FUNCTION RFID_Get_String : Buffer_Error
VAR_INPUT
	Data : REFERENCE TO RFID_Tag_Data;
	Num : USINT; 
END_VAR
VAR_IN_OUT
	Out : STRING[8];
END_VAR

RFID_Get_String := Get_String_From_Buffer(Num:= Num, 
											Layout:= Data.Layout, 
											Buffer:= Data.Data, 
											Out:= Out);

END_FUNCTION

(* stored: Version 1.1.0.1, ProductVersion 3.1.4024.10
   POU RFID_Get_String: Id {15e709f0-4fe0-48b8-a5fa-987abe07119d}, SpecialFunc None *)
